FUNCTION_BLOCK TcoMessengerTests EXTENDS TcoCore.TcoObject
VAR
	_category : TcoCore.eMessageCategory;
	_minLevel : TcoCore.eMessageCategory;
END_VAR

{attribute 'TcRpcEnable'}
METHOD INTERNAL Catastrophic
VAR_INPUT	
	Message : STRING(255);
END_VAR
_messenger.Catastrophic(Message);
END_METHOD

{attribute 'TcRpcEnable'}
METHOD INTERNAL Critical
VAR_INPUT
	Message : STRING(255);
END_VAR
_messenger.Critical(Message);
END_METHOD

{attribute 'TcRpcEnable'}
METHOD INTERNAL Debug
VAR_INPUT
	Message : STRING(255);
END_VAR
_messenger.Debug(Message);
END_METHOD

{attribute 'TcRpcEnable'}
METHOD INTERNAL Error
VAR_INPUT
	Message : STRING(255);
END_VAR
_messenger.Error(Message);
END_METHOD

{attribute 'TcRpcEnable'}
METHOD INTERNAL Info
VAR_INPUT
	Message : STRING(255);
END_VAR
_messenger.Info(Message);
END_METHOD

{attribute 'TcRpcEnable'}
METHOD INTERNAL Notify
VAR_INPUT
	Message : STRING(255);
END_VAR
_messenger.Notify(Message);
END_METHOD

{attribute 'TcRpcEnable'}
METHOD INTERNAL Post 
VAR_INPUT	
	Message : STRING(255);	
END_VAR
_messenger.Post(Message, _category);
END_METHOD

{attribute 'TcRpcEnable'}
METHOD INTERNAL Programming
VAR_INPUT
	Message : STRING(255);
END_VAR
_messenger.Programming(Message);
END_METHOD

{attribute 'TcRpcEnable'}
METHOD INTERNAL Resume
Context.Environment.Messaging.Resume();
END_METHOD

{attribute 'TcRpcEnable'}
METHOD INTERNAL SetMinLevel
Context.Environment.Messaging.MinLevel := _minLevel;
END_METHOD

{attribute 'TcRpcEnable'}
METHOD INTERNAL Suspend
Context.Environment.Messaging.Suspend();
END_METHOD

{attribute 'TcRpcEnable'}
METHOD INTERNAL TimedOut
VAR_INPUT
	Message : STRING(255);
END_VAR
_messenger.Warning(Message);
END_METHOD

{attribute 'TcRpcEnable'}
METHOD INTERNAL Trace
VAR_INPUT
	Message : STRING(255);
END_VAR
_messenger.Trace(Message);
END_METHOD

{attribute 'TcRpcEnable'}
METHOD INTERNAL Warning
VAR_INPUT
	Message : STRING(255);
END_VAR
_messenger.Warning(Message);
END_METHOD

END_FUNCTION_BLOCK

(* stored: Version 1.1.0.1
   POU TcoMessengerTests: Id {d87e08d3-1876-01a7-16f8-c33755c3cedd}, SpecialFunc None
   Method Catastrophic: Id {093578d4-4883-02db-1234-cd38a177e6a9}
   Method Critical: Id {cc04394e-ff89-0912-0edc-b599a0c7d07c}
   Method Debug: Id {d279de92-cd96-029d-39a9-f59f29b03fe7}
   Method Error: Id {8cdb9a84-d1f9-0d5c-21aa-e984960b0322}
   Method Info: Id {c925a1ca-2a19-0552-0bb5-9de32cfb972b}
   Method Notify: Id {32b9cbb6-6207-0f35-1241-0cd0d8f3e2c6}
   Method Post: Id {aa4eba68-8e3e-0790-14e4-37c20eb0fa3d}
   Method Programming: Id {ad9b3a9b-2e3a-01d3-03b2-0966d6f79bec}
   Method Resume: Id {82062340-d28d-08df-1727-1ea7f90e73d2}
   Method SetMinLevel: Id {14062f88-3c36-0c8f-1769-35d9d0ae9a98}
   Method Suspend: Id {009042cd-d9d8-01ec-1e53-e01d1459f156}
   Method TimedOut: Id {df75203d-ff31-0992-037d-6d10558ac6d6}
   Method Trace: Id {02a9dc17-bef6-0f75-27b7-d7639e83bf18}
   Method Warning: Id {032a7c5b-ea22-0043-0563-7ca4d7b308c3} *)
